 					IF Dump.DONE = TRUE THEN 
						LocalDumpActive := FALSE;
						Dump.EN := FALSE; 
						DumpingRunOutTMR_TON (IN := FALSE);
					END_IF
					//ChargingRunOutTMR_TON (IN := FALSE);
				//Start up procedure run*******************************************	
					//HMI Input TO Charger SP
					IF HMI_DB.PeakChargerSP > 10 THEN
						HMI_DB.PeakChargerSP := 10;
						ELSIF HMI_DB.PeakChargerSP <= 0 THEN
							HMI_DB.PeakChargerSP := 0;
					END_IF
					IF HMI_DB.SustChargerSP > 10 THEN 
						HMI_DB.SustChargerSP := 10;
						ELSIF HMI_DB.SustChargerSP <= 0 THEN
							HMI_DB.SustChargerSP := 0;
					END_IF
					IF HMI_DB.FormChargerSP > 35 THEN 
						HMI_DB.FormChargerSP := 35;
						ELSIF HMI_DB.FormChargerSP <= 0 THEN
							HMI_DB.FormChargerSP := 0;
					END_IF	
					IF HMI_DB.PreFormChargerSP > 30 THEN 
						HMI_DB.PreFormChargerSP := 30;
						ELSIF HMI_DB.PreFormChargerSP <= 0 THEN
							HMI_DB.PreFormChargerSP := 0;
					END_IF	
					IF HMI_DB.FormTrigChargerSP > 50 THEN 
						HMI_DB.FormTrigChargerSP := 50;
						ELSIF HMI_DB.FormTrigChargerSP <= 0 THEN
							HMI_DB.FormTrigChargerSP := 0;
					END_IF	
					IF HMI_DB.PreFormTrigChargerSP > 30 THEN 
						HMI_DB.PreFormTrigChargerSP := 30;
						ELSIF HMI_DB.PreFormTrigChargerSP <= 0 THEN
							HMI_DB.PreFormTrigChargerSP := 0;
					END_IF				
					//char 1 - 3 is peaking, 4 - 6 sust, 7 - 8 form, gls 3 is preform
					MCP_IO.Charger[1].voltageSP := HMI_DB.PeakChargerSP * 1000;
					MCP_IO.Charger[2].voltageSP := HMI_DB.PeakChargerSP * 1000;
					MCP_IO.Charger[3].voltageSP := HMI_DB.PeakChargerSP * 1000;
					MCP_IO.Charger[4].voltageSP := HMI_DB.SustChargerSP * 1000;
					MCP_IO.Charger[5].voltageSP := HMI_DB.SustChargerSP * 1000;
					MCP_IO.Charger[6].voltageSP := HMI_DB.SustChargerSP * 1000;			
					MCP_IO.Charger[7].voltageSP := HMI_DB.FormChargerSP * 1000;
					MCP_IO.Charger[8].voltageSP := HMI_DB.FormChargerSP * 1000;	
					MCP_IO.GLS3_voltageSP := HMI_DB.PreFormChargerSP * 1000;
					MCP_IO.GLS1_voltageSP := HMI_DB.FormTrigChargerSP * 1000;
					MCP_IO.GLS2_voltageSP := HMI_DB.PreFormTrigChargerSP * 1000;
					
					IF HMI_DB.CloseAllChargeRlyPB = TRUE AND Trips_DB.NoFaultDetected = TRUE AND Permissives_DB.AllChargerHVisON = FALSE AND Permissives_DB.AllChargerInhibited = TRUE THEN
						FOR j := 1 TO 3 BY 1 DO 
							//CLOSE all charge relays
							LCP.Section[j].Peak.CloseChargeRelay1 := TRUE; 
							LCP.Section[j].Peak.CloseChargeRelay2 := TRUE; 
							LCP.Section[j].Sust.CloseChargeRelay1 := TRUE;
							LCP.Section[j].Sust.CloseChargeRelay2 := TRUE;
						END_FOR;
						//CLOSE all charge rly on form
						LCP.Section[4].Form.CloseChargeRelay1 := TRUE;
						LCP.Section[4].Form.CloseChargeRelay2 := TRUE;
						LCP.Section[4].Form.CloseFormTrigChargeRly := TRUE;
						LCP.Section[4].Form.ClosePreFormChargeRly := TRUE;
						LCP.Section[4].Form.ClosePreFormTrigChargeRly := TRUE;
					ELSE
						FOR j := 1 TO 3 BY 1 DO 
							//Open all charge relays
							LCP.Section[j].Peak.CloseChargeRelay1 := FALSE; 
							LCP.Section[j].Peak.CloseChargeRelay2 := FALSE; 
							LCP.Section[j].Sust.CloseChargeRelay1 := FALSE;
							LCP.Section[j].Sust.CloseChargeRelay2 := FALSE;
						END_FOR;
						//open all charge rly on form
						LCP.Section[4].Form.CloseChargeRelay1 := FALSE;
						LCP.Section[4].Form.CloseChargeRelay2 := FALSE;
						LCP.Section[4].Form.CloseFormTrigChargeRly := FALSE;
						LCP.Section[4].Form.ClosePreFormChargeRly := FALSE;
						LCP.Section[4].Form.ClosePreFormTrigChargeRly := FALSE;	
					END_IF;
					
					//OPEN DUMP
					IF HMI_DB.OpenAllDumpRlyPB = TRUE AND Trips_DB.NoFaultDetected = TRUE AND Permissives_DB.AllChargerHVisON = FALSE AND Permissives_DB.AllChargerInhibited = TRUE THEN
						FOR j := 1 TO 3 BY 1 DO 
							//open all dump relays  - for SAFE STATE they can all go together
							LCP.Section[j].Peak.OpenDumpRelay1 := TRUE;
							LCP.Section[j].Peak.OpenDumpRelay2 := TRUE;
							LCP.Section[j].Sust.OpenDumpRelay1 := TRUE;
							LCP.Section[j].Sust.OpenDumpRelay2 := TRUE;	
						END_FOR;	
						//close all dump relay on form
						LCP.Section[4].Form.OpenDumpRelay1 := TRUE;
						LCP.Section[4].Form.OpenDumpRelay2 := TRUE;
						LCP.Section[4].Form.OpenPreFormDumpRly := TRUE;
						LCP.Section[4].Form.OpenFormTrigDumpRly1 := TRUE;
						LCP.Section[4].Form.OpenPreFormTrigDumpRly1 := TRUE;					
					ELSE
						FOR j := 1 TO 3 BY 1 DO 
							//open all dump relays  - for SAFE STATE they can all go together
							LCP.Section[j].Peak.OpenDumpRelay1 := FALSE;
							LCP.Section[j].Peak.OpenDumpRelay2 := FALSE;
							LCP.Section[j].Sust.OpenDumpRelay1 := FALSE;
							LCP.Section[j].Sust.OpenDumpRelay2 := FALSE;	
						END_FOR;	
						//close all dump relay on form
						LCP.Section[4].Form.OpenDumpRelay1 := FALSE;
						LCP.Section[4].Form.OpenDumpRelay2 := FALSE;
						LCP.Section[4].Form.OpenPreFormDumpRly := FALSE;
						LCP.Section[4].Form.OpenFormTrigDumpRly1 := FALSE;
						LCP.Section[4].Form.OpenPreFormTrigDumpRly1 := FALSE;	
					END_IF;
					
					IF HMI_DB.LiftMachineGNDsw = TRUE AND Trips_DB.NoFaultDetected = TRUE THEN
						MCP_IO.LiftMachineGND := TRUE;
						ELSE
							MCP_IO.LiftMachineGND := FALSE;
					END_IF;
					// no fault, safety ok, charger HV is OFF and Inhibited condition before opening dump relays
					IF Trips_DB.NoFaultDetected = TRUE AND 
						Permissives_DB.SafetyOK = TRUE AND
						Permissives_DB.AllPeakChargerHVisON = FALSE AND 
						Permissives_DB.AllPeakChargerInhibited = TRUE AND 
						HMI_DB.OpenAllPeakDumpRlySW = TRUE 
						THEN
							FOR j := 1 TO 3 BY 1 DO 
								//open all peak dump relays 
								LCP.Section[j].Peak.OpenDumpRelay1 := TRUE;
								LCP.Section[j].Peak.OpenDumpRelay2 := TRUE;	
							END_FOR;
						ELSIF HMI_DB.OpenAllPeakDumpRlySW = FALSE THEN
								FOR j := 1 TO 3 BY 1 DO 
									LCP.Section[j].Peak.OpenDumpRelay1 := FALSE;
									LCP.Section[j].Peak.OpenDumpRelay2 := FALSE;	
								END_FOR;
					END_IF

					IF Trips_DB.NoFaultDetected = TRUE AND 
						Permissives_DB.SafetyOK = TRUE AND
						Permissives_DB.AllSustChargerHVisON = FALSE AND 
						Permissives_DB.AllSustChargerInhibited = TRUE AND 
						HMI_DB.OpenAllSustDumpRlySW = TRUE 
						THEN
							FOR j := 1 TO 3 BY 1 DO 
								//open all sust dump relays 
								LCP.Section[j].Sust.OpenDumpRelay1 := TRUE;
								LCP.Section[j].Sust.OpenDumpRelay2 := TRUE;	
							END_FOR;
						ELSIF HMI_DB.OpenAllSustDumpRlySW = FALSE THEN 
								FOR j := 1 TO 3 BY 1 DO 
									LCP.Section[j].Sust.OpenDumpRelay1 := FALSE;
									LCP.Section[j].Sust.OpenDumpRelay2 := FALSE;	
								END_FOR;							
					END_IF
					
					IF Trips_DB.NoFaultDetected = TRUE AND 
						Permissives_DB.SafetyOK = TRUE AND
						Permissives_DB.AllFormChargerHVisON = FALSE AND 
						Permissives_DB.AllFormChargerInhibited = TRUE AND 
						HMI_DB.OpenAllFormDumpRlySW = TRUE 
						THEN
							//open all form dump relays 
							LCP.Section[4].Form.OpenDumpRelay1 := TRUE;
							LCP.Section[4].Form.OpenDumpRelay2 := TRUE;	
						ELSIF HMI_DB.OpenAllFormDumpRlySW = FALSE THEN 
								LCP.Section[4].Form.OpenDumpRelay1 := FALSE;
								LCP.Section[4].Form.OpenDumpRelay2 := FALSE;								
					END_IF					
					// preform dump
					IF Trips_DB.NoFaultDetected = TRUE AND 
						Permissives_DB.SafetyOK = TRUE AND
						LCP.Section[4].Form.PreFormChargeRly_close = FALSE AND //charge relays open
						HMI_DB.OpenAllPreFormDumpRlySW = TRUE 
						THEN
							//OPEN ALL preform dump relay
							LCP.Section[4].Form.OpenPreFormDumpRly := TRUE;
						ELSIF HMI_DB.OpenAllPreFormDumpRlySW = FALSE THEN  
								LCP.Section[4].Form.OpenPreFormDumpRly := FALSE;
					END_IF;
					
					//preform trig dump 
					IF Trips_DB.NoFaultDetected = TRUE AND 
						Permissives_DB.SafetyOK = TRUE AND
						LCP.Section[4].Form.PreFormTrigChargeRly_close = FALSE AND //charge relays open
						HMI_DB.OpenPreFormTrigDumpRlySW = TRUE 
						THEN
							//OPEN ALL preform trig dump relay
							LCP.Section[4].Form.OpenPreFormTrigDumpRly1 := TRUE;
						ELSIF HMI_DB.OpenPreFormTrigDumpRlySW = FALSE THEN
								LCP.Section[4].Form.OpenPreFormTrigDumpRly1 := FALSE;
					END_IF;					
					//form  trig dump 
					IF Trips_DB.NoFaultDetected = TRUE AND 
						Permissives_DB.SafetyOK = TRUE AND
						LCP.Section[4].Form.FormTrigChargeRly_close = FALSE AND //charge relays open
						HMI_DB.OpenFormTrigDumpRlySW = TRUE 
						THEN					
							LCP.Section[4].Form.OpenFormTrigDumpRly1 := TRUE;
						ELSIF HMI_DB.OpenFormTrigDumpRlySW = FALSE THEN
							LCP.Section[4].Form.OpenFormTrigDumpRly1 := FALSE;
					END_IF;
					
					//Charge relays
					//peak charge 
					IF Trips_DB.NoFaultDetected = TRUE AND 
						Permissives_DB.SafetyOK = TRUE AND
						Permissives_DB.AllPeakChargerHVisON = FALSE AND 
						Permissives_DB.AllPeakChargerInhibited = TRUE AND 
						Permissives_DB.AllPeakDumpRlyOpen = TRUE AND 
						HMI_DB.CloseAllPeakChargRlySW = TRUE
						THEN
							LCP.Section[1].Peak.CloseChargeRelay1 := TRUE;
							LCP.Section[1].Peak.CloseChargeRelay2 := TRUE;
							LCP.Section[2].Peak.CloseChargeRelay1 := TRUE;
							LCP.Section[2].Peak.CloseChargeRelay2 := TRUE;
							LCP.Section[3].Peak.CloseChargeRelay1 := TRUE;
							LCP.Section[3].Peak.CloseChargeRelay2 := TRUE;
						ELSIF Permissives_DB.AllPeakChargerHVisON = FALSE AND Permissives_DB.AllPeakChargerInhibited = TRUE AND HMI_DB.CloseAllPeakChargRlySW = FALSE 
							THEN
								LCP.Section[1].Peak.CloseChargeRelay1 := FALSE;
								LCP.Section[1].Peak.CloseChargeRelay2 := FALSE;
								LCP.Section[2].Peak.CloseChargeRelay1 := FALSE;
								LCP.Section[2].Peak.CloseChargeRelay2 := FALSE;
								LCP.Section[3].Peak.CloseChargeRelay1 := FALSE;
								LCP.Section[3].Peak.CloseChargeRelay2 := FALSE;
					END_IF;
					
					//sust charge
					IF Trips_DB.NoFaultDetected = TRUE AND 
						Permissives_DB.SafetyOK = TRUE AND
						Permissives_DB.AllSustChargerHVisON = FALSE AND 
						Permissives_DB.AllSustChargerInhibited = TRUE AND 
						Permissives_DB.AllSustDumpRlyOpen = TRUE AND 
						HMI_DB.CloseAllSustChargRlySW = TRUE
						THEN
							LCP.Section[1].Sust.CloseChargeRelay1 := TRUE;
							LCP.Section[1].Sust.CloseChargeRelay2 := TRUE;
							LCP.Section[2].Sust.CloseChargeRelay1 := TRUE;
							LCP.Section[2].Sust.CloseChargeRelay2 := TRUE;
							LCP.Section[3].Sust.CloseChargeRelay1 := TRUE;
							LCP.Section[3].Sust.CloseChargeRelay2 := TRUE;
						ELSIF Permissives_DB.AllSustChargerHVisON = FALSE AND Permissives_DB.AllSustChargerInhibited = TRUE AND HMI_DB.CloseAllSustChargRlySW = FALSE 
							THEN
								LCP.Section[1].Sust.CloseChargeRelay1 := FALSE;
								LCP.Section[1].Sust.CloseChargeRelay2 := FALSE;
								LCP.Section[2].Sust.CloseChargeRelay1 := FALSE;
								LCP.Section[2].Sust.CloseChargeRelay2 := FALSE;
								LCP.Section[3].Sust.CloseChargeRelay1 := FALSE;
								LCP.Section[3].Sust.CloseChargeRelay2 := FALSE;
					END_IF;
					
					//Form charge
					IF Trips_DB.NoFaultDetected = TRUE AND 
						Permissives_DB.SafetyOK = TRUE AND
						Permissives_DB.AllFormChargerHVisON = FALSE AND 
						Permissives_DB.AllFormChargerInhibited = TRUE AND 
						Permissives_DB.AllFormDumpRlyOpen = TRUE AND 
						HMI_DB.CloseAllFormChargRlySW = TRUE
						THEN
							LCP.Section[4].Form.CloseChargeRelay1 := TRUE;
							LCP.Section[4].Form.CloseChargeRelay2 := TRUE;
						ELSIF Permissives_DB.AllFormChargerHVisON = FALSE AND Permissives_DB.AllFormChargerInhibited = TRUE AND HMI_DB.CloseAllFormChargRlySW = FALSE 
							THEN
								LCP.Section[4].Form.CloseChargeRelay1 := TRUE;
								LCP.Section[4].Form.CloseChargeRelay2 := TRUE;
					END_IF;
					
					//preform charge - gls 3
					IF Trips_DB.NoFaultDetected = TRUE AND 
						Permissives_DB.SafetyOK = TRUE AND
						MCP_IO.GLS3_hvON = FALSE AND  
						LCP.Section[4].Form.PreFormDumpRly_close = FALSE AND 
						HMI_DB.CloseAllPreFormChargRlySW = TRUE
						THEN 
							LCP.Section[4].Form.ClosePreFormChargeRly := TRUE;
						ELSIF MCP_IO.GLS3_hvON = FALSE AND HMI_DB.CloseAllPreFormChargRlySW = FALSE
							THEN
								LCP.Section[4].Form.ClosePreFormChargeRly := FALSE;
					END_IF;
					
					//preform trig charg - GLS 2
					IF Trips_DB.NoFaultDetected = TRUE AND 
						Permissives_DB.SafetyOK = TRUE AND
						MCP_IO.GLS2_hvON = FALSE AND  
						LCP.Section[4].Form.PreFormTrigDumpRly1_close = FALSE AND 
						HMI_DB.ClosePreFormTrigChargeRlySW = TRUE
						THEN 
							LCP.Section[4].Form.ClosePreFormTrigChargeRly := TRUE;
						ELSIF MCP_IO.GLS1_hvON = FALSE AND HMI_DB.ClosePreFormTrigChargeRlySW = FALSE
							THEN
								LCP.Section[4].Form.ClosePreFormTrigChargeRly := FALSE;
					END_IF;	
					
					//form trig charg - GLS 1
					IF Trips_DB.NoFaultDetected = TRUE AND 
						Permissives_DB.SafetyOK = TRUE AND
						MCP_IO.GLS1_hvON = FALSE AND 
						LCP.Section[4].Form.FormTrigDumpRly1_close = FALSE AND 
						HMI_DB.CloseFormTrigChargeRlySW = TRUE
						THEN 
							LCP.Section[4].Form.CloseFormTrigChargeRly := TRUE;
						ELSIF MCP_IO.GLS1_hvON = FALSE AND HMI_DB.CloseFormTrigChargeRlySW = FALSE
							THEN
								LCP.Section[4].Form.CloseFormTrigChargeRly := FALSE;
					END_IF;										
					//hv enable 
					//peak
					IF Trips_DB.NoFaultDetected = TRUE AND
						Permissives_DB.SafetyOK = TRUE AND 
						Permissives_DB.AllPeakChargeRlyClose = TRUE AND 
						Permissives_DB.AllPeakDumpRlyOpen = TRUE AND 
						HMI_DB.PeakHVONsw = TRUE 
						THEN 
							MCP_IO.Charger[1].HV_ON := TRUE;
							MCP_IO.Charger[1].inhibit := FALSE;
							MCP_IO.Charger[2].HV_ON := TRUE;
							MCP_IO.Charger[2].inhibit := FALSE;
							MCP_IO.Charger[3].HV_ON := TRUE;
							MCP_IO.Charger[3].inhibit := FALSE;
						ELSE
							MCP_IO.Charger[1].HV_ON := FALSE;
							MCP_IO.Charger[1].inhibit := TRUE;
							MCP_IO.Charger[2].HV_ON := FALSE;
							MCP_IO.Charger[2].inhibit := TRUE;
							MCP_IO.Charger[3].HV_ON := FALSE;
							MCP_IO.Charger[3].inhibit := TRUE;
					END_IF
					
					//sust
					IF Trips_DB.NoFaultDetected = TRUE AND
						Permissives_DB.SafetyOK = TRUE AND 
						Permissives_DB.AllSustChargeRlyClose = TRUE AND 
						Permissives_DB.AllSustDumpRlyOpen = TRUE AND 
						HMI_DB.SustHVONsw = TRUE 
						THEN 
							MCP_IO.Charger[4].HV_ON := TRUE;
							MCP_IO.Charger[4].inhibit := FALSE;
							MCP_IO.Charger[5].HV_ON := TRUE;
							MCP_IO.Charger[5].inhibit := FALSE;
							MCP_IO.Charger[6].HV_ON := TRUE;
							MCP_IO.Charger[6].inhibit := FALSE;
						ELSE
							MCP_IO.Charger[4].HV_ON := FALSE;
							MCP_IO.Charger[4].inhibit := TRUE;
							MCP_IO.Charger[5].HV_ON := FALSE;
							MCP_IO.Charger[5].inhibit := TRUE;
							MCP_IO.Charger[6].HV_ON := FALSE;
							MCP_IO.Charger[6].inhibit := TRUE;
					END_IF
					
					//Form
					IF Trips_DB.NoFaultDetected = TRUE AND
						Permissives_DB.SafetyOK = TRUE AND 
						Permissives_DB.AllFormChargeRlyClose = TRUE AND 
						Permissives_DB.AllFormDumpRlyOpen = TRUE AND 
						HMI_DB.FormHVONsw = TRUE 
						THEN 
							MCP_IO.Charger[7].HV_ON := TRUE;
							MCP_IO.Charger[7].inhibit := FALSE;
							MCP_IO.Charger[8].HV_ON := TRUE;
							MCP_IO.Charger[8].inhibit := FALSE;
						ELSE
							MCP_IO.Charger[7].HV_ON := FALSE;
							MCP_IO.Charger[7].inhibit := TRUE;
							MCP_IO.Charger[8].HV_ON := FALSE;
							MCP_IO.Charger[8].inhibit := TRUE;
					END_IF
					
					//preform
					IF Trips_DB.NoFaultDetected = TRUE AND
						Permissives_DB.SafetyOK = TRUE AND 
						LCP.Section[4].Form.PreFormChargeRly_close = TRUE AND 
						LCP.Section[4].Form.PreFormDumpRly_close = FALSE AND 
						HMI_DB.PreFormHVONsw = TRUE 
						THEN 
							MCP_IO.GLS3_hvON := TRUE;
						ELSE
							MCP_IO.GLS3_hvON := FALSE;			
					END_IF
					
					//preform trig
					IF Trips_DB.NoFaultDetected = TRUE AND
						Permissives_DB.SafetyOK = TRUE AND 
						LCP.Section[4].Form.PreFormTrigChargeRly_close = TRUE AND 
						LCP.Section[4].Form.PreFormTrigDumpRly1_close = FALSE AND 
						HMI_DB.GLS2HVONsw = TRUE 
						THEN 
							MCP_IO.GLS2_hvON := TRUE;
						ELSE
							MCP_IO.GLS2_hvON := FALSE;			
					END_IF	
					
					//form trig
					IF Trips_DB.NoFaultDetected = TRUE AND
						Permissives_DB.SafetyOK = TRUE AND 
						LCP.Section[4].Form.FormTrigChargeRly_close = TRUE AND 
						LCP.Section[4].Form.FormTrigDumpRly1_close = FALSE AND 
						HMI_DB.GLS1HVONsw = TRUE 
						THEN 
							MCP_IO.GLS1_hvON := TRUE;
						ELSE
							MCP_IO.GLS1_hvON := FALSE;			
					END_IF	
					
					IF GVL.RemoteModeSelected = TRUE THEN 
						ePulseState := E_PulseState.SAFE;
					END_IF
END_CASE;


IF i > 8 THEN
	i := 1;
END_IF

IF j > 3 THEN
	j := 1;
END_IF

IF k > 8 THEN
	k := 1;
END_IF

END_PROGRAM

// ---- POUs/Dump_FB.TcPOU
FUNCTION_BLOCK Dump_FB
VAR_INPUT
	EN : BOOL;
	IN1 : BOOL; //AllCapsDischarged
	IN2 : BOOL; //AllDumpRelaysOpen
	//IN3 : BOOL; //DumpingRunOut	 
	//Heartbeat		  : BOOL;
END_VAR
VAR_OUTPUT
	DONE : BOOL;
	DumpingRunOut_Elapse : REAL;
END_VAR
VAR
	//AbortPSnRlyDelayDONE : BOOL;
	//AbortPSnRlyDelay_Timer : TON;
	//AbortPSnRlyDelay_PT : TIME;
	DumpingRunOutTMR_TON : TON;
	DumpingRunOutTMR_PT : TIME := T#190S;
	DumpingRunOutTMR_ET : TIME;
	
	i : USINT := 1;
	j : USINT := 1;
	k : USINT := 0;
END_VAR


IF EN = TRUE THEN
	//start dump runout timer
	DumpingRunOutTMR_TON (IN := TRUE, PT := DumpingRunOutTMR_PT, ET => DumpingRunOutTMR_ET);
	DumpingRunOut_Elapse := TIME_TO_REAL((DumpingRunOutTMR_PT - DumpingRunOutTMR_ET)/1000);
	//IF DumpingRunOut = TRUE AND AllCapsDischarged = TRUE AND AllDumpRelaysOpen = FALSE THEN 
	//	DONE := TRUE;
	//	ELSE 
	//		DONE := FALSE;
	//END_IF
		//	DONE := TRUE;
	//IF Heartbeat = TRUE THEN 
	//	 k := k + 1;
	//END_IF;			
	IF DumpingRunOutTMR_TON.Q = TRUE AND Permissives_DB.AllSectCapsDischarged = TRUE AND IN2 = TRUE THEN //if timer run out, and in remoter mode go to trip
		DONE := TRUE;
		DumpingRunOutTMR_TON (IN := FALSE);
		ELSE 
			DONE := FALSE; 
	END_IF
					
	//TURN OFF ALL CHARGERS
	FOR i := 1 TO 8 BY 1 DO 
		MCP_IO.Charger[i].inhibit := TRUE; 		
		MCP_IO.Charger[i].HV_ON := FALSE; 
		MCP_IO.Charger[i].voltageSP := 0;
			
		//ChargeTime_DB.ChargingTimeElapse_TON[i] (IN := FALSE); //reset charging time elapse
	END_FOR;

	MCP_IO.GLS1_hvON := FALSE;
	MCP_IO.GLS2_hvON := FALSE;
	MCP_IO.GLS3_hvON := FALSE;
	MCP_IO.GLS1_voltageSP := 0;
	MCP_IO.GLS2_voltageSP := 0;
	MCP_IO.GLS3_voltageSP := 0;
					
	//ChargeTime_DB.PreFormChargingTimeElapse_TON (IN := FALSE);
	//start delay
	//AbortPSnRlyDelay_Timer (IN := TRUE, PT := AbortPSnRlyDelay_PT);					
					
	//IF AbortPSnRlyDelay_Timer.Q = TRUE THEN 
	//	AbortPSnRlyDelayDONE := TRUE;
	//	AbortPSnRlyDelay_Timer (IN := FALSE);
	//END_IF;
					
//IF 	AbortPSnRlyDelayDONE = TRUE THEN
	FOR j := 1 TO 3 BY 1 DO 
		//Open all charge relays
		LCP.Section[j].Peak.CloseChargeRelay1 := FALSE; 
		LCP.Section[j].Peak.CloseChargeRelay2 := FALSE; 
		LCP.Section[j].Sust.CloseChargeRelay1 := FALSE;
		LCP.Section[j].Sust.CloseChargeRelay2 := FALSE;
		//close all dump relays  - for SAFE STATE they can all go together
		LCP.Section[j].Peak.OpenDumpRelay1 := FALSE;
		LCP.Section[j].Peak.OpenDumpRelay2 := FALSE;
		LCP.Section[j].Sust.OpenDumpRelay1 := FALSE;
		LCP.Section[j].Sust.OpenDumpRelay2 := FALSE;	
	END_FOR;
	//open all charge rly on form
	LCP.Section[4].Form.CloseChargeRelay1 := FALSE;
	LCP.Section[4].Form.CloseChargeRelay2 := FALSE;
	LCP.Section[4].Form.CloseFormTrigChargeRly := FALSE;
	LCP.Section[4].Form.ClosePreFormChargeRly := FALSE;
	LCP.Section[4].Form.ClosePreFormTrigChargeRly := FALSE;
	//close all dump relay on form
	LCP.Section[4].Form.OpenDumpRelay1 := FALSE;
	LCP.Section[4].Form.OpenDumpRelay2 := FALSE;
	LCP.Section[4].Form.OpenPreFormDumpRly := FALSE;
	LCP.Section[4].Form.OpenFormTrigDumpRly1 := FALSE;
	LCP.Section[4].Form.OpenPreFormTrigDumpRly1 := FALSE;
						
	//AbortPSnRlyDelay_Timer (IN := FALSE);
	//AbortPSnRlyDelayDONE := FALSE;
ELSE
	DumpingRunOutTMR_TON (IN := FALSE);
END_IF;
					
IF i > 8 THEN
	i := 1;
END_IF
					
IF j > 3 THEN
	j := 1;
END_IF

END_FUNCTION_BLOCK

// ---- POUs/ChargeTime.TcPOU
PROGRAM ChargeTime
VAR

	lca_charge_cal	 : ARRAY [1..8] OF LCA_CAL;
	i				 : INT := 1; // 1-8 instances
	j				 : INT := 1; //1 - 8 ch
	m				 : INT := 1;
	
	a				 : INT := 1; 
	
	Q				 : REAL := 1; // Charge
	Current			 : REAL := 0.1; //100mA
	
	longestChargeTime: REAL;
	
END_VAR

(*IF HMI_DB.RemoteModeSelected = FALSE THEN 
	HMI_DB.TDKLoad[1].PSratedV := 12; //veto at 10
	HMI_DB.TDKLoad[2].PSratedV := 12;
	HMI_DB.TDKLoad[3].PSratedV := 12;
	HMI_DB.TDKLoad[4].PSratedV := 12;
	HMI_DB.TDKLoad[5].PSratedV := 12;
	HMI_DB.TDKLoad[6].PSratedV := 12;
	HMI_DB.TDKLoad[7].PSratedV := 50; //veto at 35
	HMI_DB.TDKLoad[8].PSratedV := 50;
	HMI_DB.GLSLoad.PSratedV := 30;
	
	HMI_DB.TDKLoad[1].TotalCapacitance := 10000;
	HMI_DB.TDKLoad[2].TotalCapacitance := 10000;
	HMI_DB.TDKLoad[3].TotalCapacitance := 10000;
	HMI_DB.TDKLoad[4].TotalCapacitance := 16000;
	HMI_DB.TDKLoad[5].TotalCapacitance := 16000;
	HMI_DB.TDKLoad[6].TotalCapacitance := 16000;
	HMI_DB.TDKLoad[7].TotalCapacitance := 1200;
	HMI_DB.TDKLoad[8].TotalCapacitance := 1200;
	HMI_DB.GLSLoad.TotalCapacitance := 200;
	
END_IF*)

IF Recipe.PeakSupplyEN = FALSE THEN
	Recipe.TDKLoad[1].RequiredChargedV :=0;
	Setpoints.TDKLoad[1].RequiredChargedV := 0;
	Recipe.TDKLoad[2].RequiredChargedV :=0;
	Setpoints.TDKLoad[2].RequiredChargedV := 0;
	Recipe.TDKLoad[3].RequiredChargedV :=0;
	Setpoints.TDKLoad[3].RequiredChargedV := 0;
END_IF

IF Recipe.SustSupplyEN = FALSE THEN
	Recipe.TDKLoad[4].RequiredChargedV :=0;
	Setpoints.TDKLoad[4].RequiredChargedV := 0;
	Recipe.TDKLoad[5].RequiredChargedV :=0;
	Setpoints.TDKLoad[5].RequiredChargedV := 0;
	Recipe.TDKLoad[6].RequiredChargedV :=0;
	Setpoints.TDKLoad[6].RequiredChargedV := 0;
END_IF

IF Recipe.FormSupplyEN = FALSE THEN
	Recipe.TDKLoad[7].RequiredChargedV := 0;
	Setpoints.TDKLoad[7].RequiredChargedV := 0;
	Recipe.TDKLoad[8].RequiredChargedV := 0;
	Setpoints.TDKLoad[8].RequiredChargedV := 0;
END_IF

IF Recipe.PFormSupplyEN = FALSE THEN
	Recipe.GLSLoad.RequiredChargedV := 0;
	Setpoints.GLSLoad.RequiredChargedV := 0;
END_IF

//veto
//this should not happen
FOR m := 1 TO 6 BY 1 DO
	IF Setpoints.TDKLoad[m].RequiredChargedV <= -2 THEN
		Setpoints.TDKLoad[m].RequiredChargedV := -2;
	END_IF	
END_FOR

IF Setpoints.GLSLoad.RequiredChargedV <= 0 THEN
	Setpoints.GLSLoad.RequiredChargedV := 0;
END_IF	

//ch 1 - 3
IF Setpoints.TDKLoad[1].RequiredChargedV >= 10 THEN
	Setpoints.TDKLoad[1].RequiredChargedV := 10;
	ELSIF Setpoints.TDKLoad[1].RequiredChargedV < 0 THEN
		Setpoints.TDKLoad[1].RequiredChargedV := ABS(Setpoints.TDKLoad[1].RequiredChargedV); 
END_IF
IF Setpoints.TDKLoad[2].RequiredChargedV >= 10 THEN
	Setpoints.TDKLoad[2].RequiredChargedV := 10;
	ELSIF Setpoints.TDKLoad[2].RequiredChargedV < 0 THEN
		Setpoints.TDKLoad[2].RequiredChargedV := ABS(Setpoints.TDKLoad[2].RequiredChargedV); 	
END_IF
IF Setpoints.TDKLoad[3].RequiredChargedV >= 10 THEN
	Setpoints.TDKLoad[3].RequiredChargedV := 10;
	ELSIF Setpoints.TDKLoad[3].RequiredChargedV < 0 THEN
		Setpoints.TDKLoad[3].RequiredChargedV := ABS(Setpoints.TDKLoad[3].RequiredChargedV); 	
END_IF
//ch 4-6
IF Setpoints.TDKLoad[4].RequiredChargedV >= 12 THEN
	Setpoints.TDKLoad[4].RequiredChargedV := 12;
	ELSIF Setpoints.TDKLoad[4].RequiredChargedV < 0 THEN
		Setpoints.TDKLoad[4].RequiredChargedV := ABS(Setpoints.TDKLoad[4].RequiredChargedV); 	
END_IF
IF Setpoints.TDKLoad[5].RequiredChargedV >= 12 THEN
	Setpoints.TDKLoad[5].RequiredChargedV := 12;
	ELSIF Setpoints.TDKLoad[5].RequiredChargedV < 0 THEN
		Setpoints.TDKLoad[5].RequiredChargedV := ABS(Setpoints.TDKLoad[5].RequiredChargedV); 	
END_IF
IF Setpoints.TDKLoad[6].RequiredChargedV >= 12 THEN
	Setpoints.TDKLoad[6].RequiredChargedV := 12;
	ELSIF Setpoints.TDKLoad[6].RequiredChargedV < 0 THEN
		Setpoints.TDKLoad[6].RequiredChargedV := ABS(Setpoints.TDKLoad[6].RequiredChargedV); 	
END_IF
//ch 7 - 8
IF Setpoints.TDKLoad[7].RequiredChargedV >= 35 THEN
	Setpoints.TDKLoad[7].RequiredChargedV := 35;
	ELSIF Setpoints.TDKLoad[7].RequiredChargedV <= 0  THEN
		Setpoints.TDKLoad[7].RequiredChargedV := 0; 	
END_IF
IF Setpoints.TDKLoad[8].RequiredChargedV >= 35 THEN
	Setpoints.TDKLoad[8].RequiredChargedV := 35;
	ELSIF Setpoints.TDKLoad[8].RequiredChargedV <= 0 THEN
		Setpoints.TDKLoad[8].RequiredChargedV := ABS(Setpoints.TDKLoad[8].RequiredChargedV); 	
END_IF
IF Setpoints.GLSLoad.RequiredChargedV >= 30 THEN
	Setpoints.GLSLoad.RequiredChargedV := 30;
	ELSIF Setpoints.GLSLoad.RequiredChargedV <= 0 THEN
		Setpoints.GLSLoad.RequiredChargedV := 0; 	
END_IF

//mapping hmi input to setpoints
FOR j := 1 TO 8 BY 1 DO	
	Setpoints.TDKLoad[j].TotalCapacitance	:= HMI_DB.TDKLoad[j].TotalCapacitance;
	Setpoints.TDKLoad[j].PSratedV 			:= HMI_DB.TDKLoad[j].PSratedV;
	//Setpoints.PeakBank[m].RequiredChargedV	:= Recipe.PeakBank[m].RequiredChargedV; //only thing that comes from the main plc recipe
	Setpoints.TDKLoad[j].wLCA				:= HMI_DB.TDKLoad[j].wLCA;
	Setpoints.TDKLoad[j].NumOfCharger		:= HMI_DB.TDKLoad[j].NumOfCharger;	
	
	Setpoints.TDKLoad[j].TotalCapacitance	:= HMI_DB.TDKLoad[j].TotalCapacitance;
	Setpoints.TDKLoad[j].PSratedV 			:= HMI_DB.TDKLoad[j].PSratedV;
	//Setpoints.SustBank[m].RequiredChargedV	:= Recipe.SustBank[m].RequiredChargedV; //only thing that comes from the main plc recipe
	Setpoints.TDKLoad[j].wLCA				:= HMI_DB.TDKLoad[j].wLCA;
	Setpoints.TDKLoad[j].NumOfCharger		:= HMI_DB.TDKLoad[j].NumOfCharger;	
	//charge time delay and elapse for HMI
	ChargeTime_DB.ChargeTimeStartDelay[j] := TIME_TO_INT((ChargeTime_DB.ChargerDelay_PT[j] - ChargeTime_DB.ChargerDelay_ET[j])/1000);
	ChargeTime_DB.ChargingTimeElapse[j] := TIME_TO_INT((ChargeTime_DB.ChargingTimeElapse_TON[j].PT - ChargeTime_DB.ChargingTimeElapse_TON[j].ET)/1000);
END_FOR

ChargeTime_DB.PreFormChargeTimeStartDelay := TIME_TO_INT((ChargeTime_DB.PreFormChargeTime_PT - ChargeTime_DB.PreFormChargeTime_ET)/1000);
ChargeTime_DB.PreFormChargingTimeElapse := TIME_TO_INT((ChargeTime_DB.PreFormChargingTimeElapse_TON.PT - ChargeTime_DB.PreFormChargingTimeElapse_TON.ET)/1000);

//GLS 3
Setpoints.GLSLoad.TotalCapacitance	:= HMI_DB.GLSLoad.TotalCapacitance;
Setpoints.GLSLoad.PSratedV 			:= HMI_DB.GLSLoad.PSratedV;
//Setpoints.PreFormBank.RequiredChargedV	:= Recipe.PreFormBank.RequiredChargedV; //only thing that comes from the main plc recipe
//Setpoints.GLSLoad.wLCA				:= HMI_DB.GLSLoad.wLCA;
Setpoints.GLSLoad.NumOfCharger		:= HMI_DB.GLSLoad.NumOfCharger;	

//chg time
FOR i := 1 TO 8 BY 1 DO
	lca_charge_cal[i](	PSratedV := Setpoints.TDKLoad[i].PSratedV, 
						RequiredChargeV := Setpoints.TDKLoad[i].RequiredChargedV, 
						LoadCapacitance := Setpoints.TDKLoad[i].TotalCapacitance, 
						NumOfCharger := Setpoints.TDKLoad[i].NumOfCharger, 
						wLCA := Setpoints.TDKLoad[i].wLCA
						);

	MCP_IO.Charger[i].ChargeTime.timeToChargeLoad := lca_charge_cal[i].TimeToChargeLoad;
	MCP_IO.Charger[i].ChargeTime.Power := lca_charge_cal[i].RespectedPower;
END_FOR


//gls - gls3 is preform cap charger
Q := 1000* Setpoints.GLSLoad.RequiredChargedV * (Setpoints.GLSLoad.TotalCapacitance / 1000000);
MCP_IO.GLS3_Load.timeToChargeLoad := Q / Current;
MCP_IO.GLS3_Load.Power := 1000*Setpoints.GLSLoad.RequiredChargedV * Current;

//find the longest charge time.  //need more work
longestChargeTime := MAX( MCP_IO.Charger[1].ChargeTime.timeToChargeLoad,
							MCP_IO.Charger[2].ChargeTime.timeToChargeLoad,
							MCP_IO.Charger[3].ChargeTime.timeToChargeLoad,
							MCP_IO.Charger[4].ChargeTime.timeToChargeLoad,
							MCP_IO.Charger[5].ChargeTime.timeToChargeLoad,
							MCP_IO.Charger[6].ChargeTime.timeToChargeLoad,
							MCP_IO.Charger[7].ChargeTime.timeToChargeLoad,
							MCP_IO.Charger[8].ChargeTime.timeToChargeLoad, 
							MCP_IO.GLS3_Load.timeToChargeLoad);

ChargeTime_DB.LongestChargeTime_PT := REAL_TO_TIME (1000*longestChargeTime);

FOR a := 1 TO 8 BY 1 DO
	IF (longestChargeTime - MCP_IO.Charger[a].ChargeTime.timeToChargeLoad) >= 0 THEN
		ChargeTime_DB.ChargerDelay_PT[a] := REAL_TO_TIME (1000*(longestChargeTime - MCP_IO.Charger[a].ChargeTime.timeToChargeLoad));
		ELSE 
			ChargeTime_DB.ChargerDelay_PT[a] := REAL_TO_TIME (1000*(MCP_IO.Charger[a].ChargeTime.timeToChargeLoad - longestChargeTime));
	END_IF;		
		
	//IF (longestChargeTime - MCP_IO.Charger[a+3].ChargeTime.timeToChargeLoad) >= 0 THEN
	//	ChargeTime_DB.SustChargeTime_PT[a] := REAL_TO_TIME (1000*(longestChargeTime - MCP_IO.Charger[a+3].ChargeTime.timeToChargeLoad));	
	//END_IF;	
	
END_FOR;


(*IF (longestChargeTime - MCP_IO.Charger[7].ChargeTime.timeToChargeLoad) >= 0 THEN
	ChargeTime_DB.FormChargeTime_PT[1] := REAL_TO_TIME (1000*(longestChargeTime - MCP_IO.Charger[7].ChargeTime.timeToChargeLoad));	
END_IF;	
IF (longestChargeTime - MCP_IO.Charger[8].ChargeTime.timeToChargeLoad) >= 0 THEN
	ChargeTime_DB.FormChargeTime_PT[2] := REAL_TO_TIME (1000*(longestChargeTime - MCP_IO.Charger[8].ChargeTime.timeToChargeLoad));	
END_IF;	
*)
IF (longestChargeTime - MCP_IO.GLS3_Load.timeToChargeLoad) >= 0 THEN
		ChargeTime_DB.PreFormChargeTime_PT := REAL_TO_TIME (1000*(longestChargeTime - MCP_IO.GLS3_Load.timeToChargeLoad));
		ELSE
			ChargeTime_DB.PreFormChargeTime_PT := REAL_TO_TIME (1000*(MCP_IO.GLS3_Load.timeToChargeLoad -longestChargeTime));
END_IF;



IF i > 8 THEN 
	i := 0;
END_IF

IF j > 8 THEN
	j := 0;
END_IF

IF m > 6 THEN
	m := 0;
END_IF

IF a > 8 THEN 
	a := 1;
END_IF;

END_PROGRAM

// ---- POUs/Communication.TcPOU
PROGRAM Communication
VAR
	//ePulseState : E_PulseState;
	i : INT := 1; //1-3
	j : INT := 1; //1-10
	k : INT := 1; //1-12
	m : INT := 1;
	n : INT := 1;
END_VAR

//echoing voltage feedback to main plc

FOR m := 1 TO 8 BY 1 DO
	TxMainPLC.Charger[m].VoltageFeedback := MCP_IO.Charger[m].voltageFeedback; 
	TxMainPLC.Charger[m].CurrentFeedback := MCP_IO.Charger[m].currentFeedback;
	
	//recipe to setpoints
	Setpoints.TDKLoad[m].RequiredChargedV := Recipe.TDKLoad[m].RequiredChargedV;

	TxMainPLC.Charger[m].TDKLoad.timeToChargeLoad := MCP_IO.Charger[m].ChargeTime.timeToChargeLoad;
	TxMainPLC.GLSLoad.timeToChargeLoad := MCP_IO.GLS3_Load.timeToChargeLoad;
END_FOR

Setpoints.GLS1_VSP := Recipe.GLS1_VSP;
Setpoints.GLS2_VSP := Recipe.GLS2_VSP;
Setpoints.GLSLoad.RequiredChargedV := Recipe.GLSLoad.RequiredChargedV;
	
FOR i := 1 TO 3 BY 1 DO
//still needs work here.
	FOR j := 1 TO 10 BY 1 DO
		TxMainPLC.Section[i].PeakCap[j].voltageFeedback := LCP.Section[i].Peak.Cap[j].voltageFeedback;
		TxMainPLC.Section[i].PeakCap[j].currentFeedback := LCP.Section[i].Peak.Cap[j].currentFeedback;
	END_FOR;
	
	TxMainPLC.Section[i].SustCap[1].voltageFeedback := LCP.Section[i].Sust.Cap[1].voltageFeedback;
	TxMainPLC.Section[i].SustCap[1].currentFeedback := LCP.Section[i].Sust.Cap[1].currentFeedback;
	TxMainPLC.Section[i].SustCap[2].voltageFeedback := LCP.Section[i].Sust.Cap[2].voltageFeedback;
	TxMainPLC.Section[i].SustCap[2].currentFeedback := LCP.Section[i].Sust.Cap[2].currentFeedback;
	
END_FOR;

FOR k := 1 TO 12 BY 1 DO 
	TxMainPLC.Section[4].FormCap[k].voltageFeedback := LCP.Section[4].Form.Cap[k].voltageFeedback;
	TxMainPLC.Section[4].FormCap[k].currentFeedback := LCP.Section[4].Form.Cap[k].currentFeedback;
END_FOR

TxMainPLC.Section[4].FormTrigVoltage := LCP.Section[4].FormTriggerVoltageFeedback;
TxMainPLC.Section[4].PreFormTrigVoltage := LCP.Section[4].PreFormTriggerVoltageFeedback;
TxMainPLC.Section[4].PreFormCapVoltage := LCP.Section[4].PreFormCapVoltageFeedback;

TxMainPLC.ChargingRunOutTime := TIME_TO_REAL ((ChargeTime_DB.LongestChargeTime_PT + HMI_DB.RunOutTMR_PT)/1000);
TxMainPLC.ChargeRunOutTime := TIME_TO_REAL (HMI_DB.RunOutTMR_PT/1000);

IF i > 3 THEN
	i := 1;
END_IF

IF j > 10 THEN
	j := 1;
END_IF

IF k > 12 THEN
	k := 1;
END_IF

IF m > 8 THEN
	m := 1;
END_IF;


(*
FB_ReadAdsSymByName (
			bRead		:= TRUE, // on or off
			sNetID		:= 5.104.224.86.1.333, //AmsNetID
			nPort		:= 852, // plc port
			sVarName	:= E_Command,  //read from
			nDestAddr	:= E_Command, //write to 
			nLen		:= 2, //2 bytes	
			);

FB_WriteAdsSymByName (
			bWrite		:= TRUE,
			sNetID		:= 5.1.121.21.21.2,
			nPort		:= 851,
			sVarName	:= E_Status,
			nSrcAddr	:= E_Status,
			nLen		:= 2, //2byte
			);

*)

END_PROGRAM

// ---- POUs/AnalogConversion.TcPOU
PROGRAM AnalogConversion
VAR
	i					: INT := 1; //charger 1-8
	j					: INT := 1;  // section 1 - 4 
	k					: INT := 1;  // cap 1-10
	m					: INT := 1; //form cap 1-12
END_VAR

//Converting raw data into Voltage Reading (0-10V), (0.5-4.5V)   
//unfinish

//MCP Charger 
//Analog Input
FOR i := 1 TO 8 BY 1 DO
	
	MCP_IO.Charger[i].ChargerType_12kV := NOT MCP_IO.Charger[i].ChargerType_50kV;
	//voltage
	MCP_IO.Charger[i].voltageFeedback_norm := Norm_x (raw_input := INT_TO_REAL (MCP_IO.Charger[i].voltageFeedback_raw),
														x_max := 32767,
														x_min := 0);
	//current																									
	MCP_IO.Charger[i].currentFeedback_norm := Norm_x (raw_input := INT_TO_REAL (MCP_IO.Charger[i].currentFeedback_raw),
														x_max := 32767,
														x_min := 0);
	//50kV chargers feedback
	//if 50kV config selected
	IF MCP_IO.Charger[i].ChargerType_50kV = TRUE THEN 
		//50kv
		MCP_IO.Charger[i].voltageFeedback := (EngVal.Max_50kVChargerVoltage - EngVal.Min_50kVChargerVoltage) * ADC_10V(
																							normal_input := MCP_IO.Charger[i].voltageFeedback_norm,
																							x_max := 10,
																							x_min := 0);

		MCP_IO.Charger[i].currentFeedback := (EngVal.Max_50kVChargerCurrent - EngVal.Min_50kVChargerCurrent) * ADC_10V(
																							normal_input := MCP_IO.Charger[i].currentFeedback_norm,
																							x_max := 10,
																							x_min := 0);
		//12kv
	ELSIF MCP_IO.Charger[i].ChargerType_12kV = TRUE THEN
		MCP_IO.Charger[i].voltageFeedback := (EngVal.Max_12kVChargerVoltage - EngVal.Min_12kVChargerVoltage) * ADC_10V(
																							normal_input := MCP_IO.Charger[i].voltageFeedback_norm,
																							x_max := 10,
																							x_min := 0);
		MCP_IO.Charger[i].currentFeedback := (EngVal.Max_12kVChargerCurrent - EngVal.Min_12kVChargerCurrent) * ADC_10V(
																							normal_input := MCP_IO.Charger[i].currentFeedback_norm,
																							x_max := 10,
																							x_min := 0);										
	END_IF;	
END_FOR;

//Analog Output
//voltageSP = Required Charge Voltage******************
//limit for charing the cap
FOR i := 1 TO 8 BY 1 DO
	
	//if 50kV config selected
	IF MCP_IO.Charger[i].ChargerType_50kV = TRUE THEN 
		//set limits of charger voltage input 
		IF MCP_IO.Charger[i].voltageSP >= REAL_TO_DINT (EngVal.UpperLimit50kVCaps) THEN
			MCP_IO.Charger[i].voltageSP := 35000; //limit at 35kV
		ELSIF MCP_IO.Charger[i].voltageSP <= 0 THEN
			MCP_IO.Charger[i].voltageSP := 0; //limit at 0V
		END_IF; 
		
	//prepare output signal for 50kV chargers.
		MCP_IO.Charger[i].voltageSP_norm := Norm_x (raw_input := DINT_TO_REAL (MCP_IO.Charger[i].voltageSP), 
												x_max := EngVal.Max_50kVChargerVoltage,
												x_min := EngVal.Min_50kVChargerVoltage);	
												
		MCP_IO.Charger[i].voltageSP_raw := AQ (norm_input := MCP_IO.Charger[i].voltageSP_norm, 
												x_max := 10,
												x_min := 0);
	END_IF;
		
	//if 12kV config selected
	IF MCP_IO.Charger[i].ChargerType_12kV = TRUE THEN
		//set limits of charger voltage input 
		IF MCP_IO.Charger[i].voltageSP <= 0 THEN
			MCP_IO.Charger[i].voltageSP := ABS(MCP_IO.Charger[i].voltageSP);
		END_IF
		
		IF MCP_IO.Charger[i].voltageSP >= REAL_TO_DINT (EngVal.UpperLimit12kVCaps) THEN
			MCP_IO.Charger[i].voltageSP := 10000; //limit at 10kV
		END_IF;

		//prepare output signal for 12kV chargers.
		MCP_IO.Charger[i].voltageSP_norm := Norm_x (raw_input := DINT_TO_REAL (MCP_IO.Charger[i].voltageSP), 
												x_max := EngVal.Max_12kVChargerVoltage,
												x_min := EngVal.Min_12kVChargerVoltage);
		
		MCP_IO.Charger[i].voltageSP_raw := AQ (norm_input := MCP_IO.Charger[i].voltageSP_norm, 
												x_max := 10,
												x_min := 0); 
	END_IF;	
												
	//limite for output sigal (<= 10V)  this should not happen
	IF MCP_IO.Charger[i].voltageSP_raw >= 32767 THEN 
		MCP_IO.Charger[i].voltageSP_raw := 32767; 										
	END_IF;
	
END_FOR;

//limits for gls 
IF MCP_IO.GLS1_voltageSP >= REAL_TO_DINT (EngVal.Max_GLS1_ChargerV) THEN 
	MCP_IO.GLS1_voltageSP := REAL_TO_DINT (EngVal.Max_GLS1_ChargerV);
	ELSIF MCP_IO.GLS1_voltageSP <= 0 THEN
		MCP_IO.GLS1_voltageSP := 0;
END_IF
IF MCP_IO.GLS2_voltageSP >= REAL_TO_DINT (EngVal.Max_GLS2_ChargerV) THEN 
	MCP_IO.GLS2_voltageSP := REAL_TO_DINT (EngVal.Max_GLS2_ChargerV);
	ELSIF MCP_IO.GLS2_voltageSP <= 0 THEN
		MCP_IO.GLS2_voltageSP := 0 ; 
END_IF
IF MCP_IO.GLS3_voltageSP >= REAL_TO_DINT (EngVal.ULimit_PreFormCapRequiredV) THEN 
	MCP_IO.GLS3_voltageSP := REAL_TO_DINT (EngVal.ULimit_PreFormCapRequiredV);
	ELSIF MCP_IO.GLS3_voltageSP <= 0 THEN
		MCP_IO.GLS3_voltageSP := 0 ; 
END_IF

//prepare analog output for gls chargers.	
MCP_IO.GLS1_voltageSP_norm := Norm_x (raw_input := DINT_TO_REAL (MCP_IO.GLS1_voltageSP),
									x_max := EngVal.Max_GLS1_ChargerV,
									x_min := 0);
MCP_IO.GLS1_voltageSP_raw:= AQ (norm_input := MCP_IO.GLS1_voltageSP_norm,
									x_max := 10,
									x_min := 0);									
									
MCP_IO.GLS2_voltageSP_norm := Norm_x (raw_input := DINT_TO_REAL (MCP_IO.GLS2_voltageSP),
									x_max := EngVal.Max_GLS2_ChargerV,
									x_min := 0);
MCP_IO.GLS2_voltageSP_raw:= AQ (norm_input := MCP_IO.GLS2_voltageSP_norm,
									x_max := 10,
									x_min := 0);	
									
MCP_IO.GLS3_voltageSP_norm := Norm_x (raw_input := DINT_TO_REAL (MCP_IO.GLS3_voltageSP),
									x_max := EngVal.Max_GLS3_ChargerV,
									x_min := 0);
MCP_IO.GLS3_voltageSP_raw:= AQ (norm_input := MCP_IO.GLS3_voltageSP_norm,
									x_max := 10,
									x_min := 0);	

//LCP 1 - 3 AI
FOR j := 1 TO 3 BY 1 DO 
	FOR k := 1 TO 10 BY 1 DO 
		LCP.Section[j].Peak.Cap[k].voltageFeedback_Norm := Norm_x (raw_input := INT_TO_REAL (LCP.Section[j].Peak.Cap[k].voltageFeedback_raw),
																x_max := 32767,
																x_min := 0);
																
		LCP.Section[j].Peak.Cap[k].voltageFeedback := (EngVal.Max_CapVoltage - EngVal.Min_CapVoltage) * ADC_10V (
																								normal_input := LCP.Section[j].Peak.Cap[k].voltageFeedback_Norm,
																								x_max := 10,
																								x_min := 0);
		//sustain caps 1 - 2
		LCP.Section[j].Sust.Cap[1].voltageFeedback_Norm := Norm_x (raw_input := INT_TO_REAL (LCP.Section[j].Sust.Cap[1].voltageFeedback_raw),
																x_max := 32767,
																x_min := 0);
																
		LCP.Section[j].Sust.Cap[1].voltageFeedback := (EngVal.Max_CapVoltage - EngVal.Min_CapVoltage) * ADC_10V (
																								normal_input := LCP.Section[j].Sust.Cap[1].voltageFeedback_Norm,
																								x_max := 10,
																								x_min := 0);
																
		LCP.Section[j].Sust.Cap[2].voltageFeedback_Norm := Norm_x (raw_input := INT_TO_REAL (LCP.Section[j].Sust.Cap[2].voltageFeedback_raw),
																x_max := 32767,
																x_min := 0);
																
		LCP.Section[j].Sust.Cap[2].voltageFeedback := (EngVal.Max_CapVoltage - EngVal.Min_CapVoltage) * ADC_10V (
																								normal_input := LCP.Section[j].Sust.Cap[2].voltageFeedback_Norm,
																								x_max := 10,
																								x_min := 0);
	END_FOR;	
END_FOR

//LCP 4 AI
FOR m := 1 TO 12 BY 1 DO
	LCP.Section[4].Form.Cap[m].voltageFeedback_norm := Norm_x (raw_input := INT_TO_REAL (LCP.Section[4].Form.Cap[m].voltageFeedback_raw),
																x_max := 32767,
																x_min := 0);
																
	LCP.Section[4].Form.Cap[m].voltageFeedback := (EngVal.Max_CapVoltage - EngVal.Min_CapVoltage) * ADC_10V (
																							normal_input := LCP.Section[4].Form.Cap[m].voltageFeedback_norm,
																							x_max := 10,
																							x_min := 0);
END_FOR;

//preform  cap AI
LCP.Section[4].PreFormCapVoltage_norm := Norm_x (raw_input := INT_TO_REAL (LCP.Section[4].PreFormCapVoltage_raw),
														x_max := 32767,
														x_min := 0);
															
LCP.Section[4].PreFormCapVoltageFeedback := (EngVal.Max_CapVoltage - EngVal.Min_CapVoltage) * ADC_10V (
																							normal_input := LCP.Section[4].PreFormCapVoltage_norm,
																							x_max := 10,
																							x_min := 0);															


//reset counter
IF i > 8 THEN
	i:=1;
END_IF;

IF j > 3 THEN 
	j := 1;
END_IF

IF k > 10 THEN 
	k := 1;
END_IF

IF m > 12 THEN 
	m := 1;
END_IF

END_PROGRAM

// ---- POUs/HMI.TcPOU
PROGRAM HMI
VAR
END_VAR

IF MCP_IO.RemoteModeSelected = TRUE (*OR HMI_DB.RemoteModeSelected = TRUE *)THEN 
	GVL.RemoteModeSelected := TRUE;
	ELSE
//ELSIF MCP_IO.RemoteModeSelected = FALSE OR HMI_DB.RemoteModeSelected = FALSE THEN
		GVL.RemoteModeSelected := FALSE;
END_IF

END_PROGRAM

// ---- POUs/Heartbeat_1.TcPOU
PROGRAM Heartbeat_1
VAR
	start_TON				: TON;
	start_TON_et 			: TIME;
	reset_TON 				: TON;
	reset_TON_et 			: TIME;
	screen_refresh_pulse 	: BOOL;
	
	pulse_1Hz_Start_TON		: TON;
	pulse_1Hz_Start_PT		: TIME := T#500MS;
	pulse_1Hz_Reset_TON		: TON;
	pulse_1Hz_Reset_PT		: TIME := T#500MS;
	pulse_1Hz				: BOOL;
END_VAR

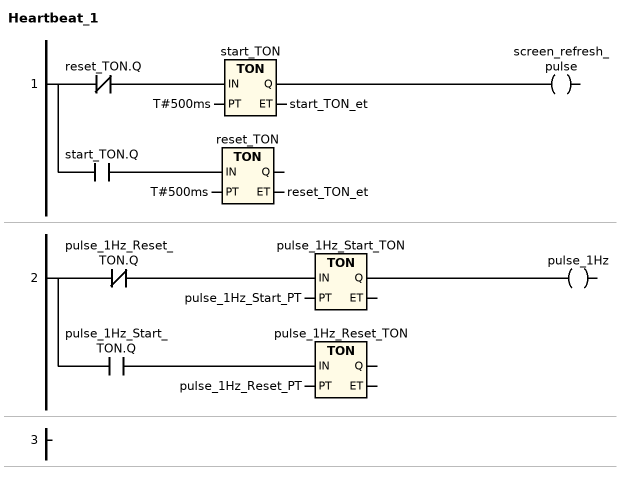
// NETWORK 1
start_TON(IN := NOT reset_TON.Q, PT := T#500ms, ET => start_TON_et); // TON
screen_refresh_pulse := start_TON.Q;
reset_TON(IN := start_TON.Q, PT := T#500ms, ET => reset_TON_et); // TON

// NETWORK 2
pulse_1Hz_Start_TON(IN := NOT pulse_1Hz_Reset_TON.Q, PT := pulse_1Hz_Start_PT); // TON
pulse_1Hz := pulse_1Hz_Start_TON.Q;
pulse_1Hz_Reset_TON(IN := pulse_1Hz_Start_TON.Q, PT := pulse_1Hz_Reset_PT); // TON

// NETWORK 3

END_PROGRAM
